FUNCTION_BLOCK E_RESTART (* Service Interface Function Block Type *)
  (* Standard: 61499-2 *)
  (* Version 0.0, 2008-07-10, 4DIAC-IDE, 4DIAC-Consortium *)
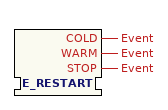
  EVENT_OUTPUT
    COLD;
    WARM;
    STOP;
  END_EVENT
  SERVICE E_RESTART/RESOURCE
    SEQUENCE cold_restart
      RESOURCE.start() -> E_RESTART.START();
    END_SEQUENCE
    SEQUENCE warm_restart
      RESOURCE.restart() -> E_RESTART.WARM();
    END_SEQUENCE
    SEQUENCE stopping
      RESOURCE.stop() -> E_RESTART.STOP();
    END_SEQUENCE
  END_SERVICE
END_FUNCTION_BLOCK
